// TwinCAT 3 PLC project Untitled1
// ProgramVersion: 3.1.4023.0
// libraries:
//   CmpBitmapPool, * (System)
//   Tc2_Standard, * (Beckhoff Automation GmbH)
//   Tc2_System, * (Beckhoff Automation GmbH)
//   Tc3_Module, * (Beckhoff Automation GmbH)
//   VisuSymbols,3.5.10.0,System
// project tree:
//   / GlobalTextList.TcGTLO, PlcTask.TcTTO, Visualization Manager.TcVMO (not stored)
//   GVLs/ DVL.TcGVL
//   POUs/ Diagram Klas.TcCD (not stored), FB_piec.TcPOU, MAIN.TcPOU
//   VISUs/ Ekran1.TcVIS
// real-time tasks:
//   TASK PlcTask: cycle T#10ms, priority 20, ADS port 350

CONFIGURATION Untitled1
    RESOURCE PLC ON TwinCAT3
        TASK PlcTask(INTERVAL := T#10ms, PRIORITY := 20);
        PROGRAM MAIN WITH PlcTask : MAIN;
    END_RESOURCE
END_CONFIGURATION

// ---- GVLs/DVL.TcGVL
{attribute 'qualified_only'}
VAR_GLOBAL
	stanprzycisku:BOOL;
END_VAR

// ---- POUs/MAIN.TcPOU
PROGRAM MAIN
VAR
    cola:FB_piec; 
    czasoOpuzniacz:TON;
END_VAR

czasoOpuzniacz(IN:=TRUE,PT:=T#10MS);
IF  czasoOpuzniacz.Q=TRUE AND DVL.stanprzycisku=TRUE THEN
    cola();
    czasoOpuzniacz(IN:=FALSE);
END_IF

END_PROGRAM

// ---- POUs/FB_piec.TcPOU
FUNCTION_BLOCK FB_piec
VAR_INPUT
END_VAR
VAR_OUTPUT
END_VAR
VAR
    stan:INT ;
    pozycjaWzdluz:INT ;
    pozycjaHoruzontalna:INT ;	
END_VAR

CASE stan OF
    0:
        IF pozycjaWzdluz<430 THEN
            pozycjaWzdluz:=pozycjaWzdluz +1;
        END_IF
        IF pozycjaWzdluz=430 THEN
            stan:=1;
        END_IF
    1:
        IF pozycjaHoruzontalna<110 THEN
            pozycjaHoruzontalna:=pozycjaHoruzontalna +1;
        END_IF
        IF pozycjaHoruzontalna = 110 THEN
            stan:=3;
        END_IF
    2:
        IF pozycjaWzdluz < 650 THEN
            pozycjaWzdluz:=pozycjaWzdluz +1;
        END_IF
        IF pozycjaWzdluz = 650 THEN
            stan:=3;
        END_IF
    3:
        metoda_Restart();

END_CASE

METHOD metoda_Restart : BOOL
VAR_INPUT
END_VAR
pozycjaWzdluz :=0;
pozycjaHoruzontalna :=0;
stan :=0;
END_METHOD

END_FUNCTION_BLOCK

// ---- GlobalTextList.TcGTLO
TEXTLIST GlobalTextList
  844 = 'Drewno'
  433 = 'Piec'
END_TEXTLIST

// ---- VISUs/Ekran1.TcVIS
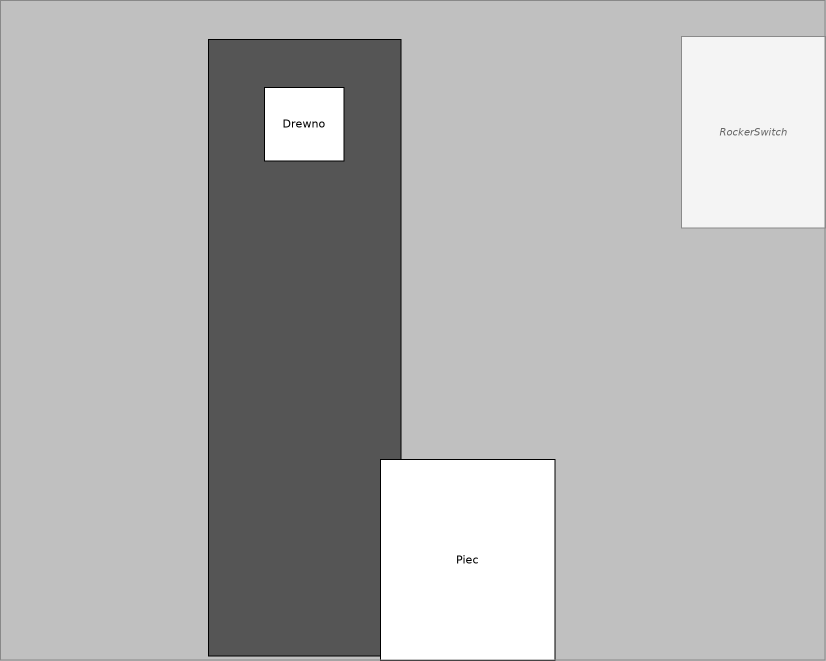
VISUALIZATION Ekran1  // 826x661
    Rectangle (208,39 193x617)
    Rectangle (264,87 80x74), "Drewno"
        p3560616238: MAIN.cola.pozycjaHoruzontalna
        p2738717112: MAIN.cola.pozycjaWzdluz
    RoundedRectangle (380,459 175x202), "Piec"
    RockerSwitch (681,36 145x192), variable: DVL.stanprzycisku, behaviour: TOGGLE, style: Switch-RockerSwitch-Gray
END_VISUALIZATION
